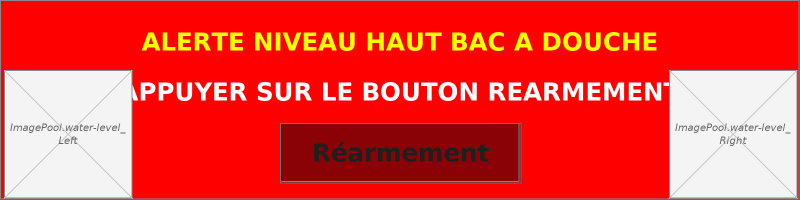
VISUALIZATION PopUp_Hight_Level  // 800x200
    Button (280,123 241x60), "Réarmement", invisible if: NOT Condi_Affich_Rearm
        OnMouseDown: toggle Cmd_Rearmement
    RoundedRectangle (0,17 800x50), "ALERTE NIVEAU HAUT BAC A DOUCHE"
    RoundedRectangle (0,67 800x50), "APPUYER SUR LE BOUTON REARMEMENT"
    Image (4,70 128x128), image: ImagePool.water-level_Left
    Image (669,70 128x128), image: ImagePool.water-level_Right
END_VISUALIZATION

(* stored: Version 1.1.0.1, ProductVersion 3.1.4024.15
   Visu PopUp_Hight_Level: Id {f61bb04a-fd8f-4022-a0be-903fa2b2531e} *)
